FUNCTION_BLOCK Konstanta (* Composite FB wrapping other FBs *)
  (* Standard: 61499-2 *)
  (* Version 1.0, 2020-08-06, Candra Wardaya, UGM *)
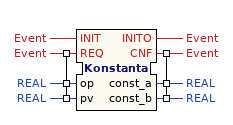
  EVENT_INPUT
    INIT; (* Initialization Request *)
    REQ WITH op, pv; (* Normal Execution Request *)
  END_EVENT
  EVENT_OUTPUT
    INITO; (* Initialization Confirm *)
    CNF WITH const_a, const_b; (* Execution Confirmation *)
  END_EVENT
  VAR_INPUT
    op : REAL; (* Controller Output Data *)
    pv : REAL; (* Process Variable Data *)
  END_VAR
  VAR_OUTPUT
    const_a : REAL; (* Constant 1 *)
    const_b : REAL; (* Constant 2 *)
  END_VAR
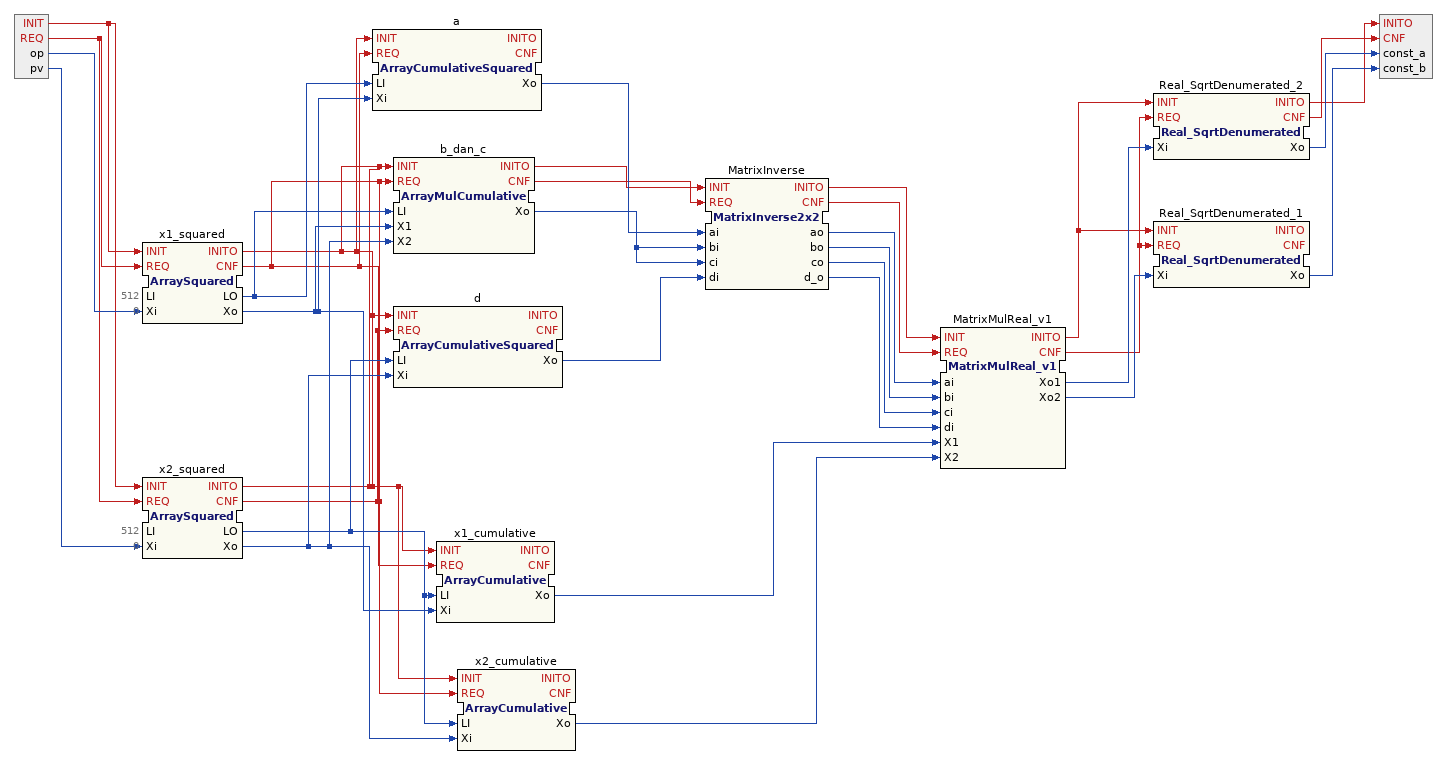
  FBS
    d : ArrayCumulativeSquared;
    x1_squared : ArraySquared(LI := 512, Xi := 0);
    MatrixMulReal_v1 : MatrixMulReal_v1;
    a : ArrayCumulativeSquared;
    x2_cumulative : ArrayCumulative;
    Real_SqrtDenumerated_1 : Real_SqrtDenumerated;
    x1_cumulative : ArrayCumulative;
    Real_SqrtDenumerated_2 : Real_SqrtDenumerated;
    x2_squared : ArraySquared(LI := 512, Xi := 0);
    b_dan_c : ArrayMulCumulative;
    MatrixInverse : MatrixInverse2x2;
  END_FBS
  EVENT_CONNECTIONS
    MatrixMulReal_v1.INITO TO Real_SqrtDenumerated_2.INIT;
    MatrixMulReal_v1.INITO TO Real_SqrtDenumerated_1.INIT;
    x1_squared.CNF TO b_dan_c.REQ;
    x1_squared.CNF TO x1_cumulative.REQ;
    x2_squared.INITO TO x2_cumulative.INIT;
    x1_squared.INITO TO a.INIT;
    x2_squared.CNF TO b_dan_c.REQ;
    x2_squared.CNF TO x2_cumulative.REQ;
    x1_squared.INITO TO x1_cumulative.INIT;
    MatrixMulReal_v1.CNF TO Real_SqrtDenumerated_1.REQ;
    x2_squared.CNF TO d.REQ;
    x2_squared.INITO TO d.INIT;
    x1_squared.INITO TO b_dan_c.INIT;
    x1_squared.CNF TO a.REQ;
    x2_squared.INITO TO b_dan_c.INIT;
    MatrixMulReal_v1.CNF TO Real_SqrtDenumerated_2.REQ;
    REQ TO x1_squared.REQ;
    INIT TO x1_squared.INIT;
    INIT TO x2_squared.INIT;
    REQ TO x2_squared.REQ;
    Real_SqrtDenumerated_2.INITO TO INITO;
    Real_SqrtDenumerated_2.CNF TO CNF;
    b_dan_c.INITO TO MatrixInverse.INIT;
    b_dan_c.CNF TO MatrixInverse.REQ;
    MatrixInverse.INITO TO MatrixMulReal_v1.INIT;
    MatrixInverse.CNF TO MatrixMulReal_v1.REQ;
  END_CONNECTIONS
  DATA_CONNECTIONS
    x2_squared.Xo TO d.Xi;
    x1_squared.Xo TO b_dan_c.X1;
    x2_squared.Xo TO x2_cumulative.Xi;
    x2_squared.Xo TO b_dan_c.X2;
    x1_squared.LO TO a.LI;
    x1_squared.Xo TO a.Xi;
    x2_squared.LO TO d.LI;
    x1_cumulative.Xo TO MatrixMulReal_v1.X1;
    x2_squared.LO TO x1_cumulative.LI;
    x2_squared.LO TO x2_cumulative.LI;
    x2_cumulative.Xo TO MatrixMulReal_v1.X2;
    x1_squared.LO TO b_dan_c.LI;
    MatrixMulReal_v1.Xo1 TO Real_SqrtDenumerated_2.Xi;
    MatrixMulReal_v1.Xo2 TO Real_SqrtDenumerated_1.Xi;
    x1_squared.Xo TO x1_cumulative.Xi;
    op TO x1_squared.Xi;
    pv TO x2_squared.Xi;
    Real_SqrtDenumerated_2.Xo TO const_a;
    Real_SqrtDenumerated_1.Xo TO const_b;
    a.Xo TO MatrixInverse.ai;
    b_dan_c.Xo TO MatrixInverse.bi;
    b_dan_c.Xo TO MatrixInverse.ci;
    d.Xo TO MatrixInverse.di;
    MatrixInverse.ao TO MatrixMulReal_v1.ai;
    MatrixInverse.bo TO MatrixMulReal_v1.bi;
    MatrixInverse.co TO MatrixMulReal_v1.ci;
    MatrixInverse.d_o TO MatrixMulReal_v1.di;
  END_CONNECTIONS
END_FUNCTION_BLOCK
